# EPICS autosave request: iocBoot/iocBasleracA130075gm/auto_settings_basler_acA1300_75gm.req
file "Basler_acA1300_75gm_settings.req",                P=$(P), R=$(R)
file "NDROI_settings.req",                              P=$(P)$(R), R=ROI1
file "NDStats_settings.req",                            P=$(P)$(R), R=Stats2
